% RSLogix 500 project AT_LAB 2 (Traffic Light).RSS, saved by version 12.00.00.00 %
PROJECT "UNTITLED"    % processor: Bul.1763 MicroLogix 1100 Series A %

PROGRAM FILES
  LAD 2   14 rungs

DATA FILES
  O0 OUTPUT  4 elements
  I1 INPUT  6 elements
  S2 STATUS  66 elements
  B3 BINARY  2 elements
  T4 TIMER  4 elements
  C5 COUNTER  1 elements
  R6 CONTROL  1 elements
  N7 INTEGER  1 elements
  F8 FLOAT  1 elements
  B30   1 elements

LADDER 2
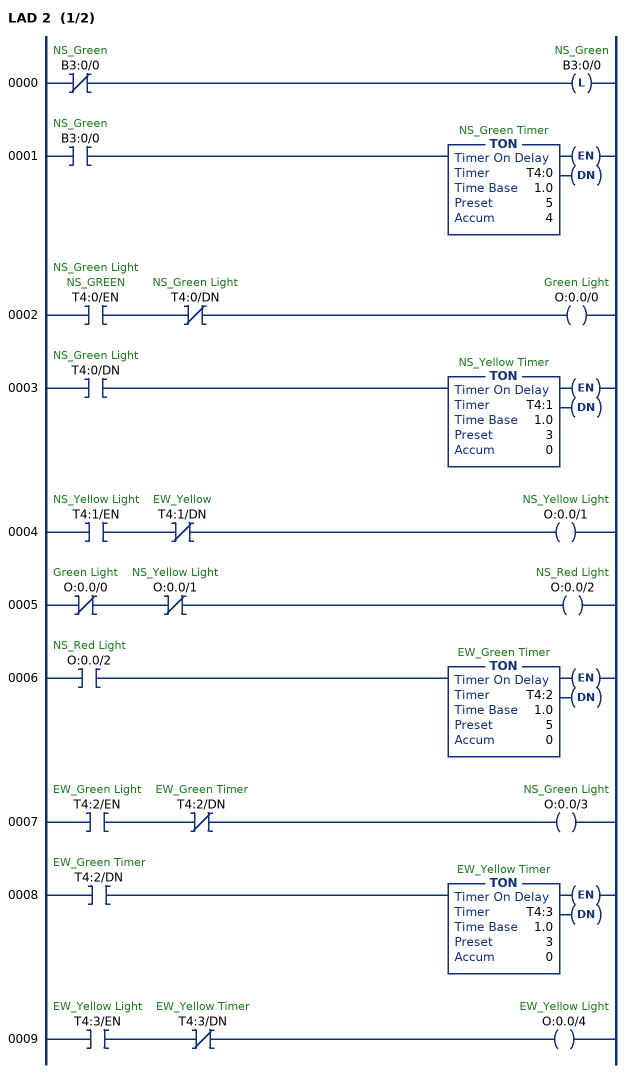
% Rung: 0 %
SOR XIO B3:0/0 OTL B3:0/0 EOR
%   B3:0/0  "NS_Green" %
% Rung: 1 %
SOR XIC B3:0/0 TON T4:0 1.0 5 4 EOR
%   B3:0/0  "NS_Green" %
%   T4:0  "NS_Green Timer" %
% Rung: 2 %
SOR XIC T4:0/EN XIO T4:0/DN OTE O:0.0/0 EOR
%   T4:0/EN  NS_GREEN  "NS_Green Light" %
%   T4:0/DN  "NS_Green Light" %
%   O:0.0/0  "Green Light" %
% Rung: 3 %
SOR XIC T4:0/DN TON T4:1 1.0 3 0 EOR
%   T4:0/DN  "NS_Green Light" %
%   T4:1  "NS_Yellow Timer" %
% Rung: 4 %
SOR XIC T4:1/EN XIO T4:1/DN OTE O:0.0/1 EOR
%   T4:1/EN  "NS_Yellow Light" %
%   T4:1/DN  "EW_Yellow" %
%   O:0.0/1  "NS_Yellow Light" %
% Rung: 5 %
SOR XIO O:0.0/0 XIO O:0.0/1 OTE O:0.0/2 EOR
%   O:0.0/0  "Green Light" %
%   O:0.0/1  "NS_Yellow Light" %
%   O:0.0/2  "NS_Red Light" %
% Rung: 6 %
SOR XIC O:0.0/2 TON T4:2 1.0 5 0 EOR
%   O:0.0/2  "NS_Red Light" %
%   T4:2  "EW_Green Timer" %
% Rung: 7 %
SOR XIC T4:2/EN XIO T4:2/DN OTE O:0.0/3 EOR
%   T4:2/EN  "EW_Green Light" %
%   T4:2/DN  "EW_Green Timer" %
%   O:0.0/3  "NS_Green Light" %
% Rung: 8 %
SOR XIC T4:2/DN TON T4:3 1.0 3 0 EOR
%   T4:2/DN  "EW_Green Timer" %
%   T4:3  "EW_Yellow Timer" %
% Rung: 9 %
SOR XIC T4:3/EN XIO T4:3/DN OTE O:0.0/4 EOR
%   T4:3/EN  "EW_Yellow Light" %
%   T4:3  "EW_Yellow Timer" %
%   O:0.0/4  "EW_Yellow Light" %

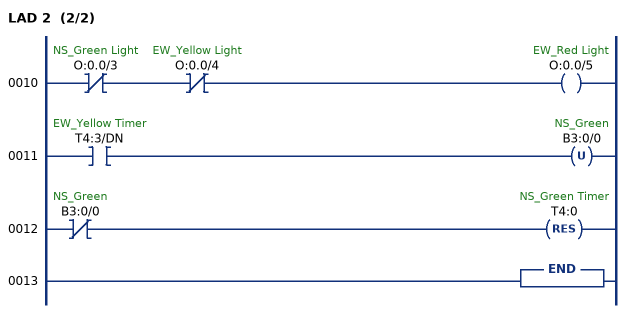
% Rung: 10 %
SOR XIO O:0.0/3 XIO O:0.0/4 OTE O:0.0/5 EOR
%   O:0.0/3  "NS_Green Light" %
%   O:0.0/4  "EW_Yellow Light" %
%   O:0.0/5  "EW_Red Light" %
% Rung: 11 %
SOR XIC T4:3/DN OTU B3:0/0 EOR
%   T4:3  "EW_Yellow Timer" %
%   B3:0/0  "NS_Green" %
% Rung: 12 %
SOR XIO B3:0/0 RES T4:0 EOR
%   B3:0/0  "NS_Green" %
%   T4:0  "NS_Green Timer" %
% Rung: 13 %
SOR END EOR

OTHER DOCUMENTED ADDRESSES
  B3:0/1  "NS_Yellow"
  I:0.0/1  "NS_Green"
  T4:0/TT  "NS_Green Light"

DATA TABLE (non-zero values as saved)
DATA B3
% B3:0 % 0X0001 0X0000
DATA T4
% .PRE .ACC %
% T4:0 % 5 4
% T4:1 % 3 0
% T4:2 % 5 0
% T4:3 % 3 0
